TYPE T_Ctrl_SIf_MOD_Cur :
STRUCT
	///[ms] time last cycle
	udiCycleTime_ms: UDINT;
END_STRUCT
END_TYPE

(* stored: Version 1.1.0.1, ProductVersion 3.1.0.18
   DUT T_Ctrl_SIf_MOD_Cur: Id {1d4d61cf-31a2-4781-8200-006aba5be2bd} *)
